FUNCTION_BLOCK PYOPCUA_CLIENT (* Basic FB with empty ECC *)
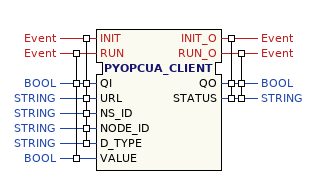
  EVENT_INPUT
    INIT WITH NODE_ID, QI, URL, NS_ID, D_TYPE;
    RUN WITH QI, VALUE;
  END_EVENT
  EVENT_OUTPUT
    INIT_O WITH STATUS, QO;
    RUN_O WITH STATUS, QO;
  END_EVENT
  VAR_INPUT
    QI : BOOL;
    URL : STRING;
    NS_ID : STRING;
    NODE_ID : STRING;
    D_TYPE : STRING;
    VALUE : BOOL;
  END_VAR
  VAR_OUTPUT
    QO : BOOL;
    STATUS : STRING;
  END_VAR
END_FUNCTION_BLOCK
